// TIA Portal project "2-Motor Conveyor System analog scaling" (V17)

(* hardware
DEVICE "S7-1200 station_1"  S7-1200 Station
   slot 0: "Rack_0"  S7-1200 Rack  Rack  V1.0
   slot 1: "PLC_1"  CPU 1214C DC/DC/DC  6ES7 214-1AG40-0XB0  V4.5
   slot 2: "AI 4x13BIT_1"  6ES7 231-4HD32-0XB0  V2.1
   slot 3: "AQ 2x14BIT_1"  SM 1232 AQ2  6ES7 232-4HB32-0XB0  V2.1
DEVICE "HMI_1"  TP700 Comfort
   slot 0: "HMI_1"  TP700 Comfort  6AV2 124-0GC01-0AX0  17.0.0.0
   slot 1: "HMI_RT_1"  TP700 Comfort  6AV2 124-0GC01-0AX0  17.0.0.0
   slot 5: "HMI_1.IE_CP_1"  PROFINET Interface  17.0.0.0
      slot 1: "PROFINET Interface_1"  PROFINET Interface
         slot 1: "Port_1"  Port
         slot 2: "Port_2"  Port
   slot 7: "HMI_1.MPI/DP_CP_1"  MPI/DP Interface  17.0.0.0
*)

// ===== PLC "PLC_1"  CPU 1214C DC/DC/DC =====

VAR_GLOBAL   // PLC tag table "Default tag table"
   "Start" AT %I0.0 : Bool;
   "Stop" AT %I0.1 : Bool;
   "Fault" AT %I0.2 : Bool;
   "Motor1_Run" AT %Q0.0 : Bool;
   "Object_detected" AT %I0.3 : Bool;
   "Motor2_Run" AT %Q0.1 : Bool;
   "Reset" AT %I0.4 : Bool;
   "Alarm" AT %Q0.2 : Bool;
   "Tag_2" AT %IW96 : Word;
END_VAR

DATA_BLOCK "Motor_1_DB"   // DB2
{ S7_Optimized_Access := 'TRUE' }
VERSION : 0.1
// stored: InstanceOfName Motor_1
"Motor_1"
BEGIN
END_DATA_BLOCK

DATA_BLOCK "Motor_2_DB"   // DB3
{ S7_Optimized_Access := 'TRUE' }
VERSION : 0.1
// stored: InstanceOfName Motor_2
"Motor_2"
BEGIN
END_DATA_BLOCK

DATA_BLOCK "Counter_DB"   // DB4
{ S7_Optimized_Access := 'TRUE' }
VERSION : 0.1
   VAR
      Object_counter : CTU_INT;
   END_VAR
   VAR RETAIN
      Temperature : Real;
   END_VAR
   VAR
      Normalized_Value : Real;
      Temp_Wire_Break : Bool;
      Temp_Overflow : Bool;
   END_VAR
BEGIN
END_DATA_BLOCK

// folder: System blocks/Program resources

DATA_BLOCK "Sort_timer_DB"   // DB1
{ S7_Optimized_Access := 'TRUE' }
AUTHOR : Simatic
FAMILY : IEC
NAME : IEC_TMR
VERSION : 1.0
// stored: InstanceOfName IEC_TIMER
"IEC_TIMER"
BEGIN
END_DATA_BLOCK

// folder: (top level)

FUNCTION_BLOCK "Motor_1"   // FB1, LAD
{ S7_Optimized_Access := 'TRUE' }
VERSION : 0.1
   VAR_INPUT
      Start : Bool;
      Stop : Bool;
      Fault : Bool;
   END_VAR
   VAR_OUTPUT
      Motor_Run : Bool;
   END_VAR
   VAR
      Latch : Bool;
   END_VAR
BEGIN

REGION Network 1
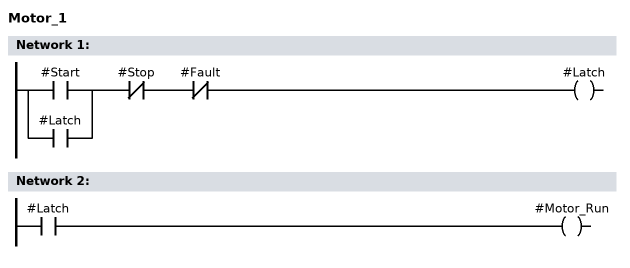
   RUNG wire#powerrail
      Contact( #Start )
      wire#w1
      I_Contact( #Stop )
      I_Contact( #Fault )
      Coil( #Latch )
   END_RUNG
   RUNG wire#powerrail
      Contact( #Latch )
   END_RUNG wire#w1
   // the same network as SCL:
   #Latch := (#Start OR #Latch) AND NOT #Stop AND NOT #Fault;
END_REGION

REGION Network 2
   RUNG wire#powerrail
      Contact( #Latch )
      Coil( #Motor_Run )
   END_RUNG
   // the same network as SCL:
   #Motor_Run := #Latch;
END_REGION
END_FUNCTION_BLOCK

FUNCTION_BLOCK "Motor_2"   // FB2, LAD
{ S7_Optimized_Access := 'TRUE' }
VERSION : 0.1
   VAR_INPUT
      Object_Detechted : Bool;
      Motor1_running : Bool;
      Stop : Bool;
      Fault : Bool;
   END_VAR
   VAR_OUTPUT
      Motor2_run : Bool;
   END_VAR
   VAR
      Sort_timer : Bool;
   END_VAR
BEGIN

REGION Network 1
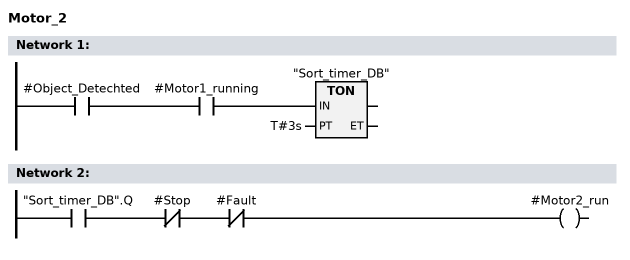
   "Sort_timer_DB".TON(IN := #Object_Detechted AND #Motor1_running, PT := T#3s);
END_REGION

REGION Network 2
   RUNG wire#powerrail
      Contact( "Sort_timer_DB".Q )
      I_Contact( #Stop )
      I_Contact( #Fault )
      Coil( #Motor2_run )
   END_RUNG
   // the same network as SCL:
   #Motor2_run := "Sort_timer_DB".Q AND NOT #Stop AND NOT #Fault;
END_REGION
END_FUNCTION_BLOCK

FUNCTION "Analog_Scaling" : Void   // FC1, SCL
{ S7_Optimized_Access := 'TRUE' }
VERSION : 0.1
   VAR_INPUT
      Raw_Value : Int;
      Eng_Min : Real;
      Eng_Max : Real;
      Raw_Min : Int;
      Raw_Max : Int;
   END_VAR
   VAR_OUTPUT
      Eng_value : Real;
      Wire_Break : Bool;
      Overflow : Bool;
   END_VAR
BEGIN
   // Wire break detection
   IF #Raw_Value < 1000 THEN
       #Wire_Break := TRUE;
       #Eng_value := 0.0;
       RETURN;
   END_IF;

   // Overflow detection  
   IF #Raw_Value > 28000 THEN
       #Overflow := TRUE;
       #Eng_value := #Eng_Max;
       RETURN;
   END_IF;

   // Normal scaling calculation
   #Wire_Break := FALSE;
   #Overflow := FALSE;

   #Eng_value := (INT_TO_REAL(#Raw_Value - #Raw_Min) *
   (#Eng_Max - #Eng_Min)) /
   INT_TO_REAL(#Raw_Max - #Raw_Min) +
   #Eng_Min;
END_FUNCTION

ORGANIZATION_BLOCK "Main"   // OB1, SCL, ProgramCycle
TITLE = "Main Program Sweep (Cycle)"
{ S7_Optimized_Access := 'TRUE' }
VERSION : 0.1
   VAR_INPUT
      Initial_Call : Bool;   // Initial call of this OB
      Remanence : Bool;   // =True, if remanent data are available
   END_VAR
BEGIN
   // ═══ MOTOR 1 — Main Conveyor Belt ═══
   "Motor_1_DB"(Start := "Start",
                Stop := "Stop",
                Fault := "Fault");

   "Motor1_Run" := "Motor_1_DB".Motor_Run;

   // ═══ MOTOR 2 — Sorting Arm ═══
   "Motor_2_DB"(Object_Detechted:="Object_detected",
                Motor1_running:="Motor_1_DB".Motor_Run,
                Stop:="Stop",
                Fault:="Fault");

   "Motor2_Run" := "Motor_2_DB".Motor2_run;

   // ═══ OBJECT COUNTER ═══
   "Counter_DB".Object_counter(
                               CU := "Object_detected",
                               R  := "Reset",
                               PV := 10);

   // ═══ AUTO STOP after 10 objects ═══
   IF "Counter_DB".Object_counter.QU THEN
       "Alarm" := TRUE; // Alarm light ON
   END_IF;

   IF "Reset" = TRUE THEN
       "Alarm" := FALSE;  // Reset alarm
   END_IF;

   "Counter_DB".Normalized_Value :=NORM_X(MIN := 0, VALUE := "Tag_2", MAX := 27648);
   "Counter_DB".Temperature := SCALE_X(MIN:=0.0, VALUE:="Counter_DB".Normalized_Value, MAX:=200.0);

   "Analog_Scaling"(
                    Raw_Value := "Tag_2",
                    Eng_Min   := 0.0,
                    Eng_Max   := 200.0,
                    Raw_Min   := 0,
                    Raw_Max   := 27648,
                    Eng_value => "Counter_DB".Temperature,
                    Wire_Break => "Counter_DB".Temp_Wire_Break,
                    Overflow   => "Counter_DB".Temp_Overflow);
END_ORGANIZATION_BLOCK

(* ===== HMI "HMI_RT_1" =====
system functions are stored by id; their names below are inferred from use
connection "HMI_Connection_1": ETHERNET, S7_1200_OMS

HMI tags "Default tag table"
   "Tag_ScreenNumber" : UInt, internal

HMI tags "Tag table_1"
   "Motor1_start" : Bool = PLC Start AT %I0.0, 1 s
   "Motor1_Stop" : Bool = PLC Stop AT %I0.1, 1 s
   "Motor1_Run" : Bool = PLC Motor1_Run AT %Q0.0, 1 s
   "Motor2_Run" : Bool = PLC Motor2_Run AT %Q0.1, 1 s
   "Object Count" : Int = PLC Counter_DB.Object_counter.CV AT %I0.3, 1 s
   "Alarm_Light" : Bool = PLC Alarm AT %Q0.2, 1 s
   "HMI_Tag_1" : Bool = PLC Alarm AT %Q0.2, 1 s
   "Temperature" : Real = PLC Counter_DB.Temperature AT %DB1.DBW0, 1 s
   "HMI_Tag_1(1)" : Real = PLC Counter_DB.Temperature, 1 s

discrete alarms
   1: '', class Warnings, trigger "HMI_Tag_1" bit 0
   2: '', class Warnings, trigger "HMI_Tag_1(1)" bit 31

screen "Root screen" 800x420, template "Template_1"
   on GenerateScreen: SetTag("Tag_ScreenNumber", 1)
   TextField "Text field_2" at 186,-2 size 344x55; Text 'Motor Conveyor System'
   Button "Button_1" at 75,58 size 96x32; TextOff 'START'
      on Click: SetBit("Motor1_start")
   Button "Button_2" at 76,112 size 96x32; TextOff 'STOP'
      on Click: ResetBit("Motor1_start"); SetBit("Motor1_Stop")
   Circle "Circle_1" at 209,58 size 83x83
      Appearance <- "Motor1_Run"
   TextField "Text field_1" at 209,144 size 96x35; Text 'MOTOR1'
   Circle "Circle_2" at 335,58 size 83x83
      Appearance <- "Motor2_Run"
   IOField "Object Counter" at 626,50 size 57x32; FormatPattern 99
      ProcessValue <- "Object Count"
   TextField "Text field_4" at 456,48 size 176x39; Text 'Objects Counted:'
   TextField "Text field_5" at 494,89 size 204x50; Text '10 Objects Reached!'
      Appearance <- "Alarm_Light"
      Visibility <- "Alarm_Light"
   Button "Button_3" at 641,364 size 74x55; TextOff 'Alarms'
      on Click: ActivateScreen("Alarm_Screen", 0)
   TextField "Text field_3" at 333,144 size 96x35; Text 'MOTOR2'
   TextField "Text field_6" at 276,207 size 197x39; Text 'Tank Temperature:'
   IOField "Object Counter_1" at 488,214 size 67x32; FormatPattern 999.9
      ProcessValue <- "Temperature"
   TextField "Text field_7" at 555,181 size 41x96; Text '°C'
   Bar "Bar_1" at 609,172 size 80x137; MinimumValue 0; MaximumValue 200
      ProcessValue <- "Temperature"

Template "Template_1" 800x420
   Button "Exit" at 720,360 size 78x58; TextOff 'Exit'; PictureOff "ExitRuntime_TP700_Comfort_TR"; PictureOn "ExitRuntime_TP700_Comfort_TR"
      on Release: StopRuntime(0)
   Button "Template_Button" at 640,360 size 78x58; TextOff 'Text'
   Button "Template_Button_1" at 560,360 size 78x58; TextOff 'Text'
   Button "Template_Button_2" at 480,360 size 78x58; TextOff 'Text'
   Button "Template_Button_3" at 400,360 size 78x58; TextOff 'Text'
   Button "Template_Button_4" at 321,360 size 78x58; TextOff 'Text'
   Button "Template_Button_5" at 241,360 size 78x58; TextOff 'Text'
   Button "Template_Button_6" at 161,360 size 78x58; TextOff 'Text'
   Button "Alarms" at 81,360 size 78x58; TextOff 'Alarms'; PictureOff "AlarmDisplay_TP700_Comfort_TR"; PictureOn "AlarmDisplay_TP700_Comfort_TR"
      on Release: function_ef3f5d25("Alarm window_Unacknowledged", -1)
   Button "Start screen" at 1,360 size 78x58; TextOff 'Start screen'; PictureOff "NavigateHome_TP700_Comfort_TR"; PictureOn "NavigateHome_TP700_Comfort_TR"
      on Release: ActivateScreen("Root screen", 0)

screen "Alarm_Screen" 800x420
   AlarmView "Alarm view_1" at 8,8 size 734x351
   Button "Button_3" at 688,368 size 76x49; TextOff 'Back'
      on Click: ActivateScreen("Root screen", 0)
*)